TYPE T_Any : __SYSTEM.AnyType; END_TYPE

(* stored: Version 1.1.0.1
   DUT T_Any: Id {2157e680-4b66-456a-90f4-593263985502} *)
